TYPE T_QueryInterface : __SYSTEM.IQueryInterface; END_TYPE

(* stored: Version 1.1.0.1, ProductVersion 3.1.4024.4
   DUT T_QueryInterface: Id {612088b5-abe5-4008-a87b-38d41d5ce749} *)
